FUNCTION_BLOCK TFCiclo_Di_Riposo_Lastre
VAR_INPUT
	Ciclo 		: POINTER TO Stato_Ciclo_Lavoro;
	Programma  : POINTER TO TFProgramma_Ciclo_Riposo_Lastre;
	ModuleAX_X : POINTER TO TFModulePalletizer_Ax;
	ModuleAX_Y : POINTER TO TFModulePalletizer_Ax;
	ModuleAX_Z : POINTER TO TFModulePalletizer_Ax;
	ModuleAX_J : POINTER TO TFModulePalletizer_AxJ_Lastre;
	StartInterpolazioneAssi : POINTER TO BOOL;
	ModulePinza : POINTER TO TFModulePalletizer_Pinza;
	QuotaPassModePuntoIntermedio : ARRAY [1..3] OF REAL;
	AbilitazioneGlobalePassMode	: BOOL;
	InterrompiCiclo : BOOL;
	Abilita_Ciclo_Step : BOOL;
	Command_Step : BOOL;
	AbilitazioneAnticipoDinamicoMovimenti : BOOL;
END_VAR
VAR_OUTPUT
	STEPDone	: BOOL;
	Errore : uint;
END_VAR
VAR
	StepInto : BOOL;
	PinzaVerticale				: BOOL;
END_VAR

(* Set della variabile che mi permette di fare lo STEP nel ciclo *)
StepInto := (Abilita_Ciclo_Step AND Command_Step) OR NOT Abilita_Ciclo_Step;

(* Reset Anticipo Dinamico se non ho l'abilitazione *)
IF NOT AbilitazioneAnticipoDinamicoMovimenti  OR NOT HMI_DisabilitaAnticipiGLOBALE THEN
	QuotaAnticipoDinamicaX_Raggiunta := FALSE;
	QuotaAnticipoDinamicaY_Raggiunta := FALSE;
	QuotaAnticipoDinamicaZ_Raggiunta := FALSE;
	QuotaAnticipoDinamicaJ_Raggiunta := FALSE;
END_IF

PinzaVerticale := ModuleAX_J^.Ax^.Status.ActPosition > 95 OR ModuleAX_J^.Ax^.Status.ActPosition < 85;

IF NOT InterrompiCiclo THEN
	IF Ciclo^.Stato = TERMINATO OR Ciclo^.Stato = ANNULLATO OR Ciclo^.Stato = INTERROTTO THEN
		 Ciclo^.Passo := 0;
	END_IF
	 Ciclo^.Stato := IN_ESECUZIONE;
	CASE  Ciclo^.Passo OF
	(* Case 0 *)
			0:   Ciclo^.Stato := IN_ESECUZIONE;
				 Ciclo^.Passo := 10;
				 Programma_Z[Z_PosFuoriIngombroRiposo].Stato 			:= NON_ESEGUITO;
				 Programma_Y[Y_PosFuoriIngombroRiposo].Stato			:= NON_ESEGUITO;
				 Programma_J[J_PosFuoriIngombro].Stato					:= NON_ESEGUITO;
				 Programma_X[X_PosDiRiposo].Stato 						:= NON_ESEGUITO;
				 Programma_Z[Z_PosDiRiposo].Stato						:= NON_ESEGUITO;
				 Programma_J[J_PosDiRiposo].Stato						:= NON_ESEGUITO;
				 
				 ProgrammaToModule_X.Stato := NON_ESEGUITO;
				 ProgrammaToModule_Y.Stato := NON_ESEGUITO;
				 ProgrammaToModule_Z.Stato := NON_ESEGUITO;
				 ProgrammaToModule_J.Stato := NON_ESEGUITO;

				 STEPDone := FALSE;
		
			(* Case 10 - Spengo aspirazione *)
			10:	IF ModulePinza^.CmdNext.Code = '' THEN
					TFParametersArrayClear(ADR(ParametersArray));
					TFCommandSend(CmdUNLOAD,ParametersArray,ModulePinza^.Cmd);
					ModulePinza^.IN.RichiestaRicalibrazioneOvemEsterna := TRUE; //Ricalibrazione automatica OVEM
					Ciclo^.Passo := 11;
				END_IF
				
			11: IF TFStateCodeGet(ModulePinza^.State) = StateUNLOAD_END THEN
					Ciclo^.Passo := 20;
				END_IF		
				
			(* Case 20 - PROGRAMMA[0] ASSE Z -> TRASLAZIONE A QUOTA DI FUORI INGOMBRO *)	
			(*
			19:	 Ciclo^.Stato := IN_ESECUZIONE;
				IF StepInto THEN
					Programma_Z[Z_PosFuoriIngombroRiposo].Stato 			:= DA_ESEGUIRE;
					Programma_Z[Z_PosFuoriIngombroRiposo].InterpolaAsse 	:= NO_INTERPOLAZIONE_ASSE;
					ProgrammaToModule_Z 									:= Programma_Z[Z_PosFuoriIngombroRiposo];
					Ciclo^.Passo := 20;
					STEPDone := FALSE;
				END_IF
				*)
			(* Case 20 - PROGRAMMA[106] ASSE Z -> TRASLAZIONE A QUOTA DI FUORI INGOMBRO *)	
			20:	
				IF StepInto THEN
					IF PinzaVerticale AND NOT AsseXInFinestraDiPrelievo THEN
						Programma_Z[Z_PosFuoriIngombroRiposo].Stato 			:= DA_ESEGUIRE;
						//Programma_Z[Z_PosFuoriIngombroRiposo].InterpolaAsse 	:= INTERPOLAZIONE_ASSE (* INTERPOLAZIONE_ASSE*);
						Programma_Z[Z_PosFuoriIngombroRiposo].InterpolaAsse 	:= No_INTERPOLAZIONE_ASSE (* INTERPOLAZIONE_ASSE*);
						ProgrammaToModule_Z 									:= Programma_Z[Z_PosFuoriIngombroRiposo];

						Programma_Y[Y_PosFuoriIngombroRiposo].Stato 			:= DA_ESEGUIRE;
						Programma_Y[Y_PosFuoriIngombroRiposo].InterpolaAsse 	:= INTERPOLAZIONE_ASSE (* INTERPOLAZIONE_ASSE*);
						ProgrammaToModule_Y 										:= Programma_Y[Y_PosFuoriIngombroRiposo];

						Programma_J[J_PosFuoriIngombro].Stato 			:= DA_ESEGUIRE;
						Programma_J[J_PosFuoriIngombro].InterpolaAsse 	:= INTERPOLAZIONE_ASSE (* INTERPOLAZIONE_ASSE*);
						ProgrammaToModule_J 							:= Programma_J[J_PosFuoriIngombro];

						StartInterpolazioneAssi^ 	:= TRUE; //Abilito l'interpolazione degli assi
					ELSE
						Programma_Z[Z_PosFuoriIngombroRiposo].Stato 			:= DA_ESEGUIRE;
						//Programma_Z[Z_PosFuoriIngombroRiposo].InterpolaAsse 	:= INTERPOLAZIONE_ASSE;
						Programma_Z[Z_PosFuoriIngombroRiposo].InterpolaAsse 	:= No_INTERPOLAZIONE_ASSE;
						ProgrammaToModule_Z 									:= Programma_Z[Z_PosFuoriIngombroRiposo];
					END_IF
					Ciclo^.Passo := 21;
					STEPDone := FALSE;
				END_IF
				
			(* Case 21 - Attesa completamento del comando MOVETOPOS o del raggiungimento quota di Pre-Movimento se abilitata la funzione*)
			21: IF (Programma_Z[Z_PosFuoriIngombroRiposo].Stato = TERMINATO OR
					Asse_Z_InFinestraDiPassMode OR 
					QuotaAnticipoDinamicaZ_Raggiunta)  AND 
					((PinzaVerticale AND NOT AsseXInFinestraDiPrelievo AND 
					(Programma_Y[Y_PosFuoriIngombroRiposo].Stato = TERMINATO OR 
					Asse_Y_InFinestraDiPassMode) AND 
					(Programma_J[J_PosFuoriIngombro].Stato = TERMINATO OR 
					Asse_J_InFinestraDiPassMode)) OR NOT PinzaVerticale OR AsseXInFinestraDiPrelievo) THEN
						Ciclo^.Passo := 24;
						STEPDone := TRUE;
				ELSIF Programma_Z[Z_PosFuoriIngombroRiposo].Stato = INTERROTTO THEN
					Ciclo^.Passo := 21;										
				END_IF
				
		(*	22: IF Programma_Z[Z_PosFuoriIngombroRiposo].Stato = INTERROTTO THEN
					 Ciclo^.Passo := 22;
				ELSIF Programma_Z[Z_PosFuoriIngombroRiposo].Stato = TERMINATO OR 
						Asse_Z_InFinestraDiPassMode OR 
						QuotaAnticipoDinamicaZ_Raggiunta THEN
							IF StepInto THEN
								Programma_J[J_PosFuoriIngombro].Stato 			:= DA_ESEGUIRE;
								Programma_J[J_PosFuoriIngombro].InterpolaAsse 	:= NO_INTERPOLAZIONE_ASSE;
								ProgrammaToModule_J		 						:= Programma_J[J_PosFuoriIngombro];
								Ciclo^.Passo := 23;
								STEPDone := FALSE;
							END_IF									
				END_IF		
			23: IF Programma_Z[Z_PosFuoriIngombroRiposo].Stato = INTERROTTO OR 
					Programma_J[J_PosFuoriIngombro].Stato = INTERROTTO THEN
					 Ciclo^.Passo := 23;
				ELSIF (Programma_Z[Z_PosFuoriIngombroRiposo].Stato = TERMINATO) AND// OR Asse_Z_InFinestraDiPassMode OR QuotaAnticipoDinamicaZ_Raggiunta) AND 
					(Programma_J[J_PosFuoriIngombro].Stato = TERMINATO OR Asse_J_InFinestraDiPassMode OR QuotaAnticipoDinamicaJ_Raggiunta) THEN
						Ciclo^.Passo := 24;
						STEPDone := TRUE;										
				END_IF	
							
				
			(* Case 24 - Scelgo in quale direzione devo muovermi per primo a seconda della disposizione delle postazioni *)	
			24:	
				CASE ASSE_DISPOSIZIONE_POSTAZIONI OF
					
					LUNGO_X:
							Ciclo^.Passo := 25;
				
					LUNGO_Y:	
							Ciclo^.Passo := 50;
			
				END_CASE
				
			(* Case 25 - Vado a quota di fuori ingombro con Y *)
			25:	IF Programma_Z[Z_PosFuoriIngombroRiposo].Stato = INTERROTTO OR
					Programma_J[J_PosFuoriIngombro].Stato = INTERROTTO THEN
						Ciclo^.Passo := 25;										
				ELSE
					IF StepInto THEN
						Programma_Y[Y_PosFuoriIngombroRiposo].Stato 			:= DA_ESEGUIRE;
						Programma_Y[Y_PosFuoriIngombroRiposo].InterpolaAsse 	:= NO_INTERPOLAZIONE_ASSE;
						ProgrammaToModule_Y 									:= Programma_Y[Y_PosFuoriIngombroRiposo];
						Ciclo^.Passo := 26;
						STEPDone := FALSE;
					END_IF
				END_IF*)

	
			(* Case 24 - Vado a quota di fuori ingombro y e j  *)
			24:
				IF Programma_Z[Z_PosFuoriIngombroRiposo].Stato = INTERROTTO OR 
					((PinzaVerticale AND NOT AsseXInFinestraDiPrelievo)AND(Programma_Y[Y_PosFuoriIngombroRiposo].Stato = INTERROTTO OR
					Programma_J[J_PosFuoriIngombro].Stato = INTERROTTO)) THEN
						Ciclo^.Passo := 24;										
				ELSE
					IF StepInto THEN
						IF (NOT PinzaVerticale AND NOT AsseXInFinestraDiPrelievo) THEN
							Programma_Y[Y_PosFuoriIngombroRiposo].Stato 			:= DA_ESEGUIRE;
							Programma_Y[Y_PosFuoriIngombroRiposo].InterpolaAsse 	:= INTERPOLAZIONE_ASSE;
							ProgrammaToModule_Y 										:= Programma_Y[Y_PosFuoriIngombroRiposo];
	
							Programma_J[J_PosFuoriIngombro].Stato 			:= DA_ESEGUIRE;
							Programma_J[J_PosFuoriIngombro].InterpolaAsse 	:= INTERPOLAZIONE_ASSE;
							ProgrammaToModule_J 							:= Programma_J[J_PosFuoriIngombro];
						END_IF
						IF NOT FuoriIngombroYNecessario THEN
							Programma_X[X_PosDiRiposo].Stato 			:= DA_ESEGUIRE;
							Programma_X[X_PosDiRiposo].InterpolaAsse 	:= INTERPOLAZIONE_ASSE;
							ProgrammaToModule_X 										:= Programma_X[X_PosDiRiposo];
							Ciclo^.Passo := 31;
						ELSE
							Ciclo^.Passo := 25;
						END_IF
						StartInterpolazioneAssi^ 	:= TRUE; //Abilito l'interpolazione degli assi
						STEPDone 					:= FALSE;
					END_IF
				END_IF
				
			(* Case 25 - *)
			25: IF Programma_Z[Z_PosFuoriIngombroRiposo].Stato = INTERROTTO OR  
					(Programma_X[X_PosDiRiposo].Stato = INTERROTTO AND NOT FuoriIngombroYNecessario) OR
					Programma_Y[Y_PosFuoriIngombroRiposo].Stato = INTERROTTO OR
					Programma_J[J_PosFuoriIngombro].Stato = INTERROTTO THEN
						Ciclo^.Passo := 25;
				ELSIF (Programma_Y[Y_PosFuoriIngombroRiposo].Stato = TERMINATO OR 
					Asse_Y_InFinestraDiPassMode) AND 
					(Programma_J[J_PosFuoriIngombro].Stato = TERMINATO OR 
					Asse_J_InFinestraDiPassMode) THEN	
						Ciclo^.Passo := 30;
						STEPDone := TRUE;									
				END_IF
					
			(* Case 26 - Check se a quota di fuori ingombro con Y *)		
			26:	IF Programma_Y[Y_PosFuoriIngombroRiposo].Stato = INTERROTTO OR 
					Programma_Z[Z_PosFuoriIngombroRiposo].Stato = INTERROTTO OR 
					Programma_J[J_PosFuoriIngombro].Stato = INTERROTTO THEN
						Ciclo^.Passo := 26;
				ELSE	
					IF Programma_Y[Y_PosFuoriIngombroRiposo].Stato = TERMINATO OR 
						Asse_Y_InFinestraDiPassMode THEN
							Ciclo^.Passo := 30;
							STEPDone := TRUE;							
					END_IF
				END_IF
										
			(* Case 30 - PROGRAMMA[0] ASSE X  -> TRASLAZIONE A QUOTA DI RIPOSO  *)	
			30:	IF Programma_Z[Z_PosFuoriIngombroRiposo].Stato = INTERROTTO OR 
					Programma_Y[Y_PosFuoriIngombroRiposo].Stato = INTERROTTO OR 
					Programma_J[J_PosFuoriIngombro].Stato = INTERROTTO THEN
						Ciclo^.Passo := 30;										
				ELSE
					IF StepInto THEN
						Programma_X[X_PosDiRiposo].Stato := DA_ESEGUIRE;
						Programma_X[X_PosDiRiposo].InterpolaAsse := NO_INTERPOLAZIONE_ASSE;
						ProgrammaToModule_X := Programma_X[X_PosDiRiposo];
					
						Ciclo^.Passo := 31;
						STEPDone := FALSE;
					END_IF
				END_IF			
				
			(* Case 31 -  Attesa completamento del comando MOVETOPOS o del raggiungimento quota di Pre-Movimento se abilitata la funzione *)
			31: 
				IF Programma_X[X_PosDiRiposo].Stato = INTERROTTO OR
					Programma_Y[Y_PosFuoriIngombroRiposo].Stato = INTERROTTO OR
					Programma_Z[Z_PosFuoriIngombroRiposo].Stato = INTERROTTO OR 
					Programma_J[J_PosFuoriIngombro].Stato = INTERROTTO THEN
						Ciclo^.Passo := 31;
				ELSE	
					IF (Programma_X[X_PosDiRiposo].Stato = TERMINATO OR Asse_X_InFinestraDiPassMode OR QuotaAnticipoDinamicaX_Raggiunta) THEN 
						Ciclo^.Passo := 32;
						STEPDone := TRUE;							
					END_IF
				END_IF
				
			(* Case 32 - Vado a quota di riposo con Y,Z,J *)
			32:
				IF Programma_X[X_PosDiRiposo].Stato = INTERROTTO OR
					Programma_Y[Y_PosFuoriIngombroRiposo].Stato = INTERROTTO OR
					Programma_Z[Z_PosFuoriIngombroRiposo].Stato = INTERROTTO OR 
					Programma_J[J_PosFuoriIngombro].Stato = INTERROTTO THEN
						Ciclo^.Passo := 32;										
				ELSE
					IF StepInto THEN
						TFParametersArrayClear(ADR(ParametersArray));
						Programma_Y[Y_PosDiRiposo].Stato := DA_ESEGUIRE;
						Programma_Y[Y_PosDiRiposo].InterpolaAsse := INTERPOLAZIONE_ASSE;
					
						Programma_Z[Z_PosDiRiposo].Stato := DA_ESEGUIRE;
						//Programma_Z[Z_PosDiRiposo].InterpolaAsse := INTERPOLAZIONE_ASSE;
						Programma_Z[Z_PosDiRiposo].InterpolaAsse := NO_INTERPOLAZIONE_ASSE;
						
						Programma_J[J_PosDiRiposo].Stato := DA_ESEGUIRE;
						Programma_J[J_PosDiRiposo].InterpolaAsse := INTERPOLAZIONE_ASSE;
						
						ProgrammaToModule_Y := Programma_Y[Y_PosDiRiposo];
						ProgrammaToModule_Z := Programma_Z[Z_PosDiRiposo];
						ProgrammaToModule_J := Programma_J[J_PosDiRiposo];
						
						StartInterpolazioneAssi^ := TRUE; //Abilito l'interpolazione degli assi
												
						Ciclo^.Passo := 90;
						STEPDone := FALSE;
					END_IF
				END_IF
												
			(* Case 50 - Vado a quota di RIPOSO con X *)
			50:	IF Programma_Z[Z_PosFuoriIngombroRiposo].Stato = INTERROTTO OR
					Programma_J[J_PosFuoriIngombro].Stato = INTERROTTO THEN
						Ciclo^.Passo := 50;										
				ELSE
					IF StepInto THEN
						Programma_X[X_PosDiRiposo].Stato 				:= DA_ESEGUIRE;
						Programma_X[X_PosDiRiposo].InterpolaAsse 		:= NO_INTERPOLAZIONE_ASSE;
						ProgrammaToModule_X 							:= Programma_X[X_PosDiRiposo];
						Ciclo^.Passo := 51;
						STEPDone := FALSE;
					END_IF
				END_IF
					
			(* Case 51 - Check se a quota di fuori RIPOSO con X *)		
			51:	IF Programma_X[X_PosDiRiposo].Stato = INTERROTTO OR 
					Programma_Z[Z_PosFuoriIngombroRiposo].Stato = INTERROTTO OR 
					Programma_J[J_PosFuoriIngombro].Stato = INTERROTTO THEN
						Ciclo^.Passo := 51;
				ELSE	
					IF Programma_X[X_PosDiRiposo].Stato = TERMINATO OR Asse_X_InFinestraDiPassMode OR QuotaAnticipoDinamicaX_Raggiunta THEN
						Ciclo^.Passo := 52;
						STEPDone := TRUE;							
					END_IF
				END_IF
												
			(* Case 52 - Vado a quota di riposo con Y,Z,J *)
			52:
				IF Programma_X[X_PosDiRiposo].Stato = INTERROTTO OR
					Programma_Z[Z_PosFuoriIngombroRiposo].Stato = INTERROTTO OR 
					Programma_J[J_PosFuoriIngombro].Stato = INTERROTTO THEN
						Ciclo^.Passo := 52;										
				ELSE
					IF StepInto THEN
						TFParametersArrayClear(ADR(ParametersArray));
						Programma_Y[Y_PosDiRiposo].Stato 			:= DA_ESEGUIRE;
						Programma_Y[Y_PosDiRiposo].InterpolaAsse 	:= INTERPOLAZIONE_ASSE;
					
						//Programma_Z[Z_PosDiRiposo].Stato 			:= DA_ESEGUIRE;
						//Programma_Z[Z_PosDiRiposo].InterpolaAsse 	:= INTERPOLAZIONE_ASSE;
						
						Programma_J[J_PosDiRiposo].Stato 			:= DA_ESEGUIRE;
						Programma_J[J_PosDiRiposo].InterpolaAsse 	:= INTERPOLAZIONE_ASSE;
						
						ProgrammaToModule_Y := Programma_Y[Y_PosDiRiposo];
						//ProgrammaToModule_Z := Programma_Z[Z_PosDiRiposo];
						ProgrammaToModule_J := Programma_J[J_PosDiRiposo];
						
						StartInterpolazioneAssi^ := TRUE; //Abilito l'interpolazione degli assi
												
						Ciclo^.Passo := 53;
						STEPDone := FALSE;
					END_IF
				END_IF

			(* Case 53 - Vado a quota di riposo con Z *)
			53:
				IF Programma_X[X_PosDiRiposo].Stato = INTERROTTO OR
					Programma_Y[Y_PosDiRiposo].Stato = INTERROTTO OR 
					Programma_J[J_PosDiRiposo].Stato = INTERROTTO THEN
						Ciclo^.Passo := 53;										
				ELSE
					IF StepInto THEN
						IF Programma_Y[Y_PosDiRiposo].Stato = TERMINATO (*OR Asse_Y_InFinestraDiPassMode)*) AND 
							Programma_J[J_PosDiRiposo].Stato = TERMINATO (*OR Asse_J_InFinestraDiPassMode)*) THEN
					
								Programma_Z[Z_PosDiRiposo].Stato 			:= DA_ESEGUIRE;
								Programma_Z[Z_PosDiRiposo].InterpolaAsse 	:= NO_INTERPOLAZIONE_ASSE;
								
								ProgrammaToModule_Z := Programma_Z[Z_PosDiRiposo];
								
								StartInterpolazioneAssi^ := FALSE; //Abilito l'interpolazione degli assi
														
								Ciclo^.Passo := 90;
								STEPDone := FALSE;
						END_IF
					END_IF
				END_IF

			(* Case 90 - Attesa completamento posizionamento di tutti gli assi *)
			90: 
				IF Programma_Y[Y_PosDiRiposo].Stato = TERMINATO (*OR Asse_Y_InFinestraDiPassMode)*) AND 
					Programma_J[J_PosDiRiposo].Stato = TERMINATO (*OR Asse_J_InFinestraDiPassMode)*) AND
					Programma_X[X_PosDiRiposo].Stato = TERMINATO (*OR Asse_X_InFinestraDiPassMode)*) AND 
					Programma_Z[Z_PosDiRiposo].Stato = TERMINATO (*OR Asse_Z_InFinestraDiPassMode)*) THEN
						Ciclo^.Passo := 1000;
						STEPDone := TRUE;
				ELSIF Programma_Y[Y_PosDiRiposo].Stato = INTERROTTO OR 
					Programma_J[J_PosDiRiposo].Stato = INTERROTTO OR 
					Programma_X[X_PosDiRiposo].Stato = INTERROTTO OR
					Programma_Z[Z_PosDiRiposo].Stato = TERMINATO THEN

						Ciclo^.Passo := 90;									
				END_IF
				
			(* Case 1000 *)
			1000:
				 Ciclo^.Stato := TERMINATO;
				 Ciclo^.Passo := 1000;
	ELSE;
	END_CASE;
ELSE								//Se il ciclo deve essere interrotto, setto il suo nuovo stato
	 Ciclo^.Stato := INTERROTTO;
END_IF

END_FUNCTION_BLOCK

(* stored: Version 1.1.0.1, ProductVersion 3.1.4024.11
   POU TFCiclo_Di_Riposo_Lastre: Id {c9e2f4b4-b199-496f-a3b9-6bdc919e5071}, SpecialFunc None *)
